// TIA Portal V20 export
VAR_GLOBAL   // PLC tag table "MCP"
   DI_PB_StartCycle AT %I128.0 : Bool;
   DI_PB_ResetAlarm AT %I128.1 : Bool;
   DI_PB_PowerOFF AT %I128.2 : Bool;
   DI_PB_ShutdownPC AT %I128.3 : Bool;
   DI_PB_LightTest AT %I128.4 : Bool;
   DI_PB_RemoteOpenShutter AT %I128.6 : Bool;
   DI_FreeI128_7 AT %I128.7 : Bool;
   DQ_AlarmBlueLED AT %Q127.1 : Bool;
   DQ_StartCycleGreenLED AT %Q127.0 : Bool;
   DQ_RemoteOpenShutterWhiteLED AT %Q127.5 : Bool;
   DQ_ShutdownPCYellowLED AT %Q127.3 : Bool;
   DQ_LightTestWhiteLED AT %Q127.4 : Bool;
   DI_PB_PowerON AT %I128.5 : Bool;
   DQ_PowerOnGreenLED AT %Q127.2 : Bool;
   DQ_FreeQ127_6 AT %Q127.6 : Bool;
   DQ_FreeQ127_7 AT %Q127.7 : Bool;
   MCP1_In AT %I118.0 : "LBP_typeMcp483StandardInput";
   MCP1_Out AT %Q120.0 : "LBP_typeMcp483StandardOutput";
END_VAR
